// Mitsubishi GX Works2 project: Class1_Relay&AND&OR   PLC: Q03UD

PROGRAM MAIN
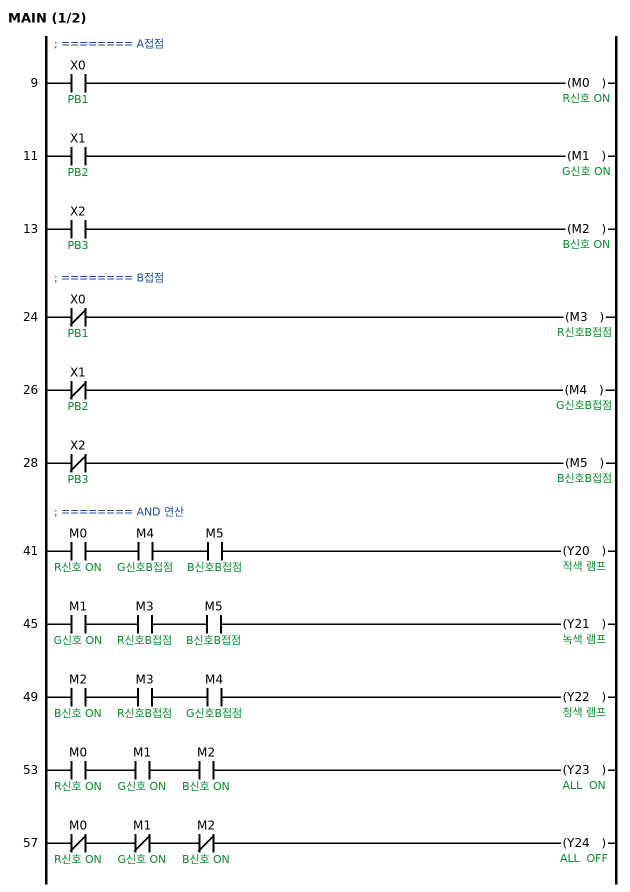
; ======== A접점
9     LD      X0  ; PB1
      OUT     M0  ; R신호 ON
11    LD      X1  ; PB2
      OUT     M1  ; G신호 ON
13    LD      X2  ; PB3
      OUT     M2  ; B신호 ON
; ======== B접점
24    LDI     X0  ; PB1
      OUT     M3  ; R신호B접점
26    LDI     X1  ; PB2
      OUT     M4  ; G신호B접점
28    LDI     X2  ; PB3
      OUT     M5  ; B신호B접점
; ======== AND 연산
41    LD      M0  ; R신호 ON
      AND     M4  ; G신호B접점
      AND     M5  ; B신호B접점
      OUT     Y20  ; 적색 램프
45    LD      M1  ; G신호 ON
      AND     M3  ; R신호B접점
      AND     M5  ; B신호B접점
      OUT     Y21  ; 녹색 램프
49    LD      M2  ; B신호 ON
      AND     M3  ; R신호B접점
      AND     M4  ; G신호B접점
      OUT     Y22  ; 청색 램프
53    LD      M0  ; R신호 ON
      AND     M1  ; G신호 ON
      AND     M2  ; B신호 ON
      OUT     Y23  ; ALL  ON
57    LDI     M0  ; R신호 ON
      ANI     M1  ; G신호 ON
      ANI     M2  ; B신호 ON
      OUT     Y24  ; ALL  OFF
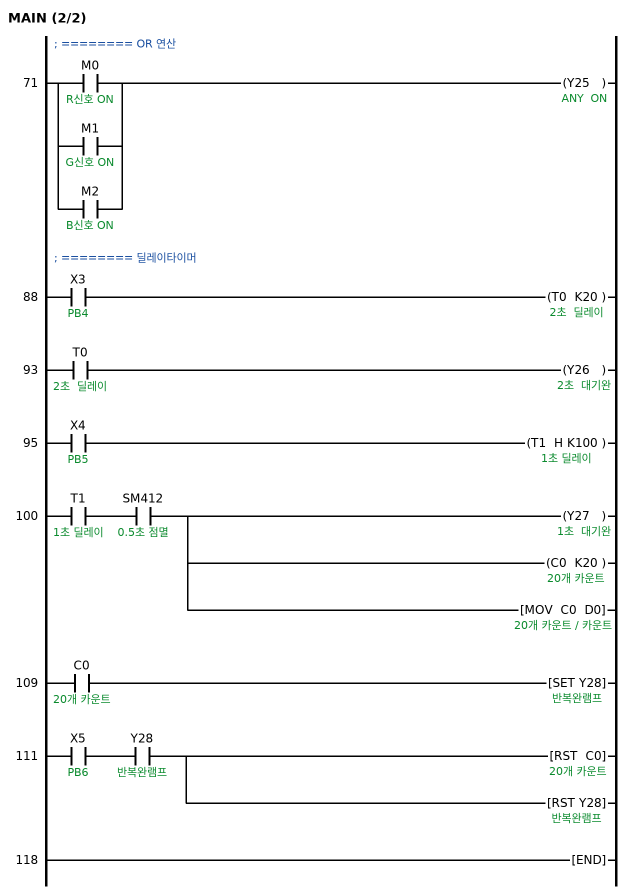
; ======== OR 연산
71    LD      M0  ; R신호 ON
      OR      M1  ; G신호 ON
      OR      M2  ; B신호 ON
      OUT     Y25  ; ANY  ON
; ======== 딜레이타이머
88    LD      X3  ; PB4
      OUT     T0 K20  ; 2초  딜레이
93    LD      T0  ; 2초  딜레이
      OUT     Y26  ; 2초  대기완
95    LD      X4  ; PB5
      OUTH    T1 K100  ; 1초 딜레이
100   LD      T1  ; 1초 딜레이
      AND     SM412  ; 0.5초 점멸
      OUT     Y27  ; 1초  대기완
      OUT     C0 K20  ; 20개 카운트
      MOV     C0 D0  ; 카운트
109   LD      C0  ; 20개 카운트
      SET     Y28  ; 반복완램프
111   LD      X5  ; PB6
      AND     Y28  ; 반복완램프
      RST     C0  ; 20개 카운트
      RST     Y28  ; 반복완램프
118   END
END_PROGRAM
